{attribute addProperty BoxType "EK1100-0000-0018"}
{attribute addProperty Id "Beckhoff_EPP3xxxEK1122Beckhoff_EPP3xxxEK1122_A4C927747992999"}
{attribute addProperty CRC "4053327647"}
{attribute addProperty SizeInBites "7992"}
{attribute addProperty SizeInBytes "999"}
TYPE Beckhoff_EPP3xxx_F198DF1F EXTENDS EK1100_179A0949 :
STRUCT
	{attribute addProperty Name "Beckhoff_EPP3xxxEK1122"}
	Beckhoff_EPP3xxxEK1122 : Beckhoff_EPP3xxxEK1122_A4C92774;
END_STRUCT
END_TYPE

(* stored: Version 1.2.0.0, ProductVersion 3.1.4024.9
   DUT Beckhoff_EPP3xxx_F198DF1F: Id {2ac4f4f8-cfd0-44fe-9265-c02d18413ede} *)
